// TwinCAT 3 PLC project Untitled1
// ProgramVersion: 3.1.4024.0
// libraries:
//   Tc2_ModbusSrv, * (Beckhoff Automation GmbH)
//   Tc2_Standard, * (Beckhoff Automation GmbH)
//   Tc2_System, * (Beckhoff Automation GmbH)
//   Tc3_Module, * (Beckhoff Automation GmbH)
// project tree:
//   / PlcTask.TcTTO
//   POUs/ MAIN.TcPOU
// real-time tasks:
//   TASK PlcTask: cycle T#10ms, priority 20, ADS port 350
//   TASK PlcTask1: cycle T#10ms, priority 21, ADS port 351

CONFIGURATION Untitled1
    RESOURCE PLC ON TwinCAT3
        TASK PlcTask(INTERVAL := T#10ms, PRIORITY := 21);
        PROGRAM MAIN WITH PlcTask : MAIN;
    END_RESOURCE
END_CONFIGURATION

// ---- POUs/MAIN.TcPOU
PROGRAM MAIN
VAR
	fbMBWriteSingleReg :FB_MBWriteSingleReg ;
	nWriteValue : INT ;
	fbTrigger : R_TRIG ;
	eWriteState : (WAIT, TRIGGER, WRITE) ;
END_VAR

fbTrigger () ;
IF fbTrigger.Q THEN
	IF eReadState = WAIT THEN
		eReadState := Trigger ;
	END_IF
END_IF
CASE eReadState 
	WAIT:
	//bişey yazılmıyor.
	
	TRIGGER :
	FB_MBWriteSingleReg(
	sIPAddr:= '127.0.0.1', 
	nTCPPort:= 502, 
	nUnitID:= 16#FF, 
	nMBAddr:= , 
	nValue:= , 
	bExecute:= , 
	tTimeout:= , 
	bBusy=> , 
	bError=> , 
	nErrId=> );
END_CASE

END_PROGRAM
